{attribute 'qualified_only'}
{attribute 'strict'}
TYPE ButtonStatus:
(
        PRESSED := 0,
        RELEASED := 1
);
END_TYPE

(* stored: Version 1.1.0.1, ProductVersion 3.1.4024.12
   DUT ButtonStatus: Id {94851a91-51ad-49a5-a978-21064361c948} *)
